{attribute 'OPC.UA.DA.StructuredType' := '1'}
TYPE ST_VSIStorageSetParameters :
STRUCT
	bLoadingAlgorithm: BOOL;
	bLoadingManual : BOOL;
END_STRUCT
END_TYPE

(* stored: Version 1.1.0.1, ProductVersion 3.1.4024.10
   DUT ST_VSIStorageSetParameters: Id {d7fbd4e5-e909-4752-a264-fe814119a1a3} *)
